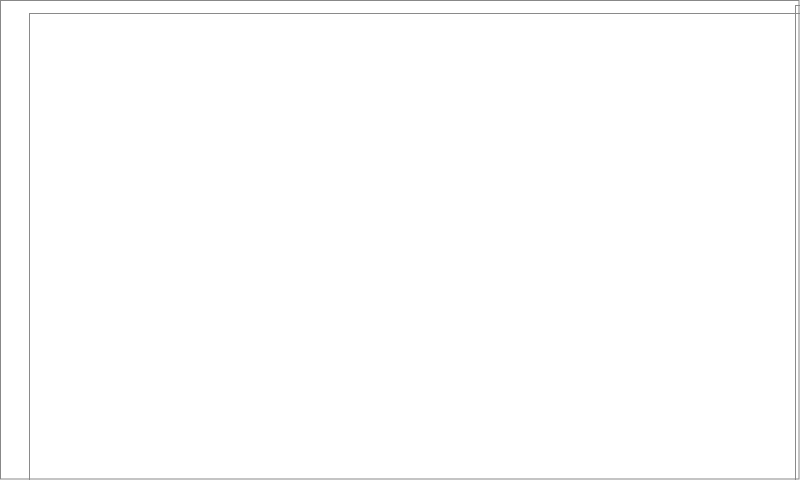
VISUALIZATION vMAIN  // 800x480
    Frame (29,13 780x996)
        shows vACTION(vACTION := ACTION1, vACTION2 := ACTION2)
    Frame (795,5 780x1000)
        shows vACTION(vACTION := ACTION1, vACTION2 := ACTION2)
    Table (37,1012 1084x201), data array: fbEventLogger.EventBuffer
        p3854506369: fbEventLogger.EventBuffer[INDEX].eEventType
        p1892666644: fbEventLogger.EventBuffer[INDEX].eEventSeverity
        p338671338: fbEventLogger.EventBuffer[INDEX].nEventIdentity
        p2170511999: fbEventLogger.EventBuffer[INDEX].sEventName
        p3723444502: fbEventLogger.EventBuffer[INDEX].sEventText
        p1218418051: fbEventLogger.EventBuffer[INDEX].dtTimestamp
END_VISUALIZATION

(* stored: Version 1.1.0.1, ProductVersion 3.1.4024.12
   Visu vMAIN: Id {4537162b-5f0d-49cf-ad43-cab00bff90cc} *)
